//enum of states
{attribute 'strict'}
{attribute 'to_string'}
{attribute 'qualified_only'}
TYPE eWsl15 :
(
	TotalReset,
	WriteFifoIntX,
	WriteFifoIntXnext,
	
	Ready,
	Error
);
END_TYPE

(* stored: Version 1.1.0.1
   DUT eWsl15: Id {61bdfcf9-0dda-41f7-bc2e-628b9dcc7323} *)
